# EPICS substitutions: apps/jscalerApp/Db/subs/jscalers_TDCFTOF1_TRIG.substitutions
file "db/jscaler_channel_DISC.db" {
pattern { CrNo,CrName,Sl,Ch,Det,Sys,Element,CScode,ThreshTDC,ThreshTRG,Mode,CountsGTDC,CountsGTRG,CountsTDC,CountsTRG,Counts }
{ "05","TDCFTOF1","20","15","TRIG","DISC","SEC1_F00","0x1405","0x110F","0x120F","0x10F","0x140F","0x130F","0x160F","0x150F","0x30F" }
}
